// TIA Portal V19 export
TYPE "LAF_typeXyzhandlingEm4Parameters"
// stored: Access Published
   STRUCT
      cm1Axis119 : "LAF_typeAxisParameters";
      cm2Axis120 { S7_SetPoint := 'True'} : "LAF_typeAxisParameters";
      cm3Axis121 { S7_SetPoint := 'True'} : "LAF_typeAxisParameters";
   END_STRUCT;
END_TYPE
